TYPE Mat4d : ARRAY[1..4, 1..4] OF LREAL; END_TYPE

(* stored: Version 1.1.0.1, ProductVersion 3.1.4024.12
   DUT Mat4d: Id {3005a4a7-d43b-43fa-bc9e-707dd33962c6} *)
